// A time instance function block that represents a date and time value based on the Unix epoch (1st Jan 1970, 00:00:00.000).
// The block provides various methods and properties to interact with the time instance, including support for UTC and local time representations.
// It can be used for time calculations, comparisons, and conversions to different time formats (e.g., `DT`, `DATE`, `TOD`).
//
// [usage]
// The time instance can be set using various methods such as `FromDateTime` or `FromEpochMilliseconds`. 
// Use properties like `Year`, `Month`, `DayOfMonth`, `Hour`, and `Minute` to extract specific components of the date and time.
// Additionally, the `ToLocal` and `ToUTC` properties allow switching between different time modes.
// Use the `Kind` property to check the time mode.
{attribute 'enable_dynamic_creation'}
{attribute 'no_explicit_call' := 'calling this function block directly is not allowed'}
FUNCTION_BLOCK FINAL FB_TimeInstance 
IMPLEMENTS 
	I_TimeInstance, I_ComparableTimesInstance, I_EquatableTimesInstance, 
	I_TimeInstanceProperties, I_TimeInstanceArithmetics, I_TimeInstanceConversions
VAR
    _nEpochMilliseconds : ULINT; // The raw time instance value in milliseconds since 1st Jan 1970.
    _Date				: SysTimeRtc.SYSTIMEDATE; // Structured representation of the time instance (year, month, day, etc.).
    _eKind				: E_TimeInstanceKind; // Indicates whether the time instance is in UTC or Local time.
END_VAR

// The day of the month extracted from the time instance.
// [get] Returns the day component of the date, with a value ranging from 1 to 31.
PROPERTY DayOfMonth : T_DayOfMonth
GET
DayOfMonth := THIS^._Date.wDay;
END_GET
END_PROPERTY

// The day of the week extracted from the time instance.
// [get] Returns the day as an `E_DayOfWeek` enum or value ranging from 1 (Monday) to 7 (Sunday).
PROPERTY DayOfWeek : E_DayOfWeek
GET
DayOfWeek := THIS^._Date.wDayOfWeek;
END_GET
END_PROPERTY

// The day of the year extracted from the time instance.
// [get] Returns the day of the year, with a value ranging from 1 to 366.
PROPERTY DayOfYear : T_DayOfYear
GET
DayOfYear := THIS^._Date.wYday;
END_GET
END_PROPERTY

// The time instance value represented as the number of milliseconds since
// Thursday, 1.1.1970 00:00:00.000 (Unix epoch).
// [get] Returns the time instance value in milliseconds.
PROPERTY EpochMilliseconds : ULINT
GET
EpochMilliseconds := THIS^._nEpochMilliseconds;
END_GET
END_PROPERTY

// Sets the time instance based on a given `DATE` value as UTC.
METHOD FromDate : I_TimeInstance // A reference to the current instance.
VAR_INPUT
	// The input `DATE` value to convert to a time instance.
	dValue : DATE;
END_VAR
VAR_OUTPUT
	// Error code indicating the result of the operation.
	Error : FsError.T_Error;
END_VAR
FromDate := THIS^;

THIS^.FromEpochMilliseconds(TO_ULINT(dValue) * 1000, Error => Error);
END_METHOD

// Sets the time instance based on a given `DT` (Date and Time) value as UTC.
METHOD FromDateTime : I_TimeInstance // A reference to the current instance.
VAR_INPUT
	// The input `DT` value to convert to a time instance.
	dtValue : DT;
END_VAR
VAR_OUTPUT
	// Error code indicating the result of the operation.
	Error : FsError.T_Error;
END_VAR
FromDateTime := THIS^;

THIS^.FromEpochMilliseconds(TO_ULINT(dtValue) * 1000, Error => Error);
END_METHOD

// Sets the time instance based on a given number of milliseconds since the Unix epoch (1st Jan 1970, 00:00:00.000).
METHOD FromEpochMilliseconds : I_TimeInstance // A reference to the current instance.
VAR_INPUT
	// The input time instance value representing the number of milliseconds since 1st Jan 1970, 00:00:00.000.
	nValue : ULINT;
END_VAR
VAR_OUTPUT
	// Error code indicating the result of the operation.
	Error : FsError.T_Error;
END_VAR
VAR
	eResult : FsError.E_CodesysCmpError;
END_VAR
FromEpochMilliseconds := THIS^;

IF THIS^._nEpochMilliseconds = nValue THEN RETURN; END_IF

eResult := SysTimeRtc.SysTimeRtcConvertHighResToDate(nValue, THIS^._Date);
CASE eResult OF
	FsError.E_CodesysCmpError.ERR_OK:
		THIS^._eKind := E_TimeInstanceKind.UTC;
		THIS^._nEpochMilliseconds := nValue;
ELSE
	Error := 
		FsError.F_CreateErrorFromStartRange(
			FsError.GVL_ErrorDescriptors.fbGeneralErrorCodes,
			FsError.E_GeneralErrorCode.ERR_CODESYS_BEGIN,
			eResult);
	THIS^.FB_init(FALSE, FALSE);
	END_CASE
END_METHOD

// Sets the time instance using the specified `LTIME` value. 
// This method converts the input value to milliseconds since the Unix epoch (1st Jan 1970, 00:00:00.000). 
//
// [note] 
// The method only considers the time value down to the millisecond precision. 
// Any values smaller than 1ms (e.g., microseconds or nanoseconds) will be ignored.
METHOD FromTime : I_TimeInstance // A reference to the current instance.
VAR_INPUT
	// The time value to be set, provided as an LTIME datatype (milliseconds since the Unix epoch).
	tValue : LTIME;
END_VAR
VAR_OUTPUT
	// Error code indicating the result of the operation.
	Error : FsError.T_Error;
END_VAR
FromTime := THIS^;

THIS^.FromEpochMilliseconds(TO_ULINT(tValue) / TO_ULINT(LTIME#1MS), Error => Error);
END_METHOD

// Sets the time instance based on a given `TOD` (Time Of Day) value as UTC.
METHOD FromTimeOfDay : I_TimeInstance // A reference to the current instance.
VAR_INPUT
	// The input `TOD` value to convert to a time instance.
	tdValue : TOD;
END_VAR
VAR_OUTPUT
	// Error code indicating the result of the operation.
	Error : FsError.T_Error;
END_VAR
FromTimeOfDay := THIS^;

THIS^.FromEpochMilliseconds(TO_ULINT(tdValue), Error => Error);
END_METHOD

// The hour of the day extracted from the time instance.
// [get] Returns the hour component of the time, with a value ranging from 0 to 23.
PROPERTY Hour : T_Hour
GET
Hour := THIS^._Date.wHour;
END_GET
END_PROPERTY

// The reference to the current time instance.
// [get] Returns a reference to the current time instance implementing `I_TimeInstance`.
PROPERTY Instance : I_TimeInstance
GET
Instance := THIS^;
END_GET
END_PROPERTY

// Checks if the current time instance is after the specified time instance.
METHOD IsAfter : BOOL // TRUE if the current time instance is after the specified one, FALSE otherwise.
VAR_INPUT
	// The time instance to compare against.
	ipOther : I_TimeInstance;
END_VAR
IsAfter := 
	ipOther <> 0
	AND_THEN
	THIS^._nEpochMilliseconds > ipOther.EpochMilliseconds;
END_METHOD

// Checks if the current time instance is before the specified time instance.
METHOD IsBefore : BOOL // TRUE if the current time instance is before the specified one, FALSE otherwise.
VAR_INPUT
	// The time instance to compare against.
	ipOther : I_TimeInstance;
END_VAR
IsBefore := 
	ipOther <> 0
	AND_THEN
	THIS^._nEpochMilliseconds < ipOther.EpochMilliseconds;
END_METHOD

// Checks if the current time instance is equal to the specified time instance.
METHOD IsEqualTo : BOOL // TRUE if the current time instance is equal to the specified, FALSE otherwise.
VAR_INPUT
	// The time instance to compare against.
	ipOther : I_TimeInstance;
END_VAR
IsEqualTo := 
	ipOther <> 0
	AND_THEN
	THIS^._nEpochMilliseconds = ipOther.EpochMilliseconds;
END_METHOD

// Specifies whether the time instance is in UTC or local time format.
// [get] Returns the time instance type enum as a value.
PROPERTY Kind : E_TimeInstanceKind
GET
Kind := THIS^._eKind;
END_GET
END_PROPERTY

// The millisecond part of the second extracted from the time instance.
// [get] Returns the millisecond component, with a value ranging from 0 to 999.
PROPERTY Millisecond : T_Millisecond
GET
Millisecond := THIS^._Date.wMilliseconds;
END_GET
END_PROPERTY

// The minute of the hour extracted from the time instance.
// [get] Returns the minute component, with a value ranging from 0 to 59.
PROPERTY Minute : T_Minute
GET
Minute := THIS^._Date.wMinute;
END_GET
END_PROPERTY

// The month of the year extracted from the time instance.
// [get] Returns the month as an `E_Month` enum or a value ranging from 1 to 12 value.
PROPERTY Month : E_Month
GET
Month := THIS^._Date.wMonth;
END_GET
END_PROPERTY

// Updates the internal epoch milliseconds of the time instance to the current system time in UTC format.
METHOD Now : REFERENCE TO FB_TimeInstance // A reference to the current instance.
VAR_OUTPUT
	// Error code indicating the result of the operation.
	Error : FsError.T_Error;
END_VAR
VAR
	eResult : FsError.E_CodesysCmpError;
END_VAR
Now REF= THIS^;

// Get the current time instance as UTC.
eResult := SysTimeRtc.SysTimeRtcHighResGet(THIS^._nEpochMilliseconds);
CASE eResult OF
	FsError.E_CodesysCmpError.ERR_OK:
		SysTimeRtc.SysTimeRtcConvertHighResToDate(THIS^._nEpochMilliseconds, THIS^._Date);
ELSE // Reset the time instance class if there's an error.
	Error := 
		FsError.F_CreateErrorFromStartRange(
			FsError.GVL_ErrorDescriptors.fbGeneralErrorCodes,
			FsError.E_GeneralErrorCode.ERR_CODESYS_BEGIN,
			eResult);
	THIS^.FB_init(FALSE, FALSE);
	END_CASE
END_METHOD

// The second of the minute extracted from the time instance.
// [get] Returns the second component, with a value ranging from 0 to 59.
PROPERTY Second : T_Second
GET
Second := THIS^._Date.wSecond;
END_GET
END_PROPERTY

// Converts the time instance to a date value.
METHOD ToDate : DATE // The date part of the time instance.
VAR_OUTPUT
	// Error code indicating the result of the operation.
	Error : FsError.T_Error;
END_VAR
ToDate := TO_DATE(THIS^.ToDateTime(Error => Error));
END_METHOD

// Converts the time instance to a combined date and time value.
METHOD ToDateTime : DT // The combined date and time value as a DT (Date and Time).
VAR_OUTPUT
	// Error code indicating the result of the operation.
	Error : FsError.T_Error;
END_VAR
VAR
	nLocal : DWORD;
	eResult : FsError.E_CodesysCmpError;
END_VAR
CASE THIS^._eKind OF
	E_TimeInstanceKind.Local:
		eResult := SysTimeRtc.SysTimeRtcConvertUtcToLocal(
			TO_DWORD(THIS^._nEpochMilliseconds / 1000),
			nLocal);
	
		ToDateTime := TO_DT(nLocal);
		
		IF eResult <> FsError.E_CodesysCmpError.ERR_OK THEN 
			Error := 
				FsError.F_CreateErrorFromStartRange(
					FsError.GVL_ErrorDescriptors.fbGeneralErrorCodes,
					FsError.E_GeneralErrorCode.ERR_CODESYS_BEGIN,
					eResult);
			END_IF
		
ELSE 
	ToDateTime := TO_DT(THIS^._nEpochMilliseconds / 1000);
	END_CASE
END_METHOD

// Converts the time instance to local time representation.
METHOD ToLocal : I_TimeInstance // A reference to the current instance.
VAR_OUTPUT
	// Error code indicating the result of the operation.
	Error : FsError.T_Error;
END_VAR
VAR
	eResult : FsError.E_CodesysCmpError;
END_VAR
ToLocal := THIS^;

IF THIS^._eKind = E_TimeInstanceKind.Local THEN RETURN; END_IF;

eResult := SysTimeRtc.SysTimeRtcConvertHighResToLocal(THIS^._nEpochMilliseconds, THIS^._Date);
CASE eResult OF
	FsError.E_CodesysCmpError.ERR_OK:
		THIS^._eKind := E_TimeInstanceKind.Local;
ELSE
	Error := 
		FsError.F_CreateErrorFromStartRange(
			FsError.GVL_ErrorDescriptors.fbGeneralErrorCodes,
			FsError.E_GeneralErrorCode.ERR_CODESYS_BEGIN,
			eResult);
	END_CASE
END_METHOD

// Converts the time instance to a time of day  value.
METHOD ToTimeOfDay : TOD // The time of day part of the time instance.
VAR_INPUT
END_VAR
ToTimeOfDay := TO_TOD(
	(THIS^._Date.wHour * TO_DWORD(TOD#01:00:00.000))
	+
	(THIS^._Date.wMinute * TO_DWORD(TOD#00:01:00.000))
	+ 
	(THIS^._Date.wSecond * TO_DWORD(TOD#00:00:01.000))
	+ 
	THIS^._Date.wMilliseconds);
END_METHOD

// Converts the time instance to UTC time representation.
METHOD ToUTC : I_TimeInstance // A reference to the current instance.
VAR_OUTPUT
	// Error code indicating the result of the operation.
	Error : FsError.T_Error;
END_VAR
VAR
	eResult : FsError.E_CodesysCmpError;
END_VAR
ToUTC := THIS^;

IF THIS^._eKind = E_TimeInstanceKind.UTC THEN RETURN; END_IF;

eResult := SysTimeRtc.SysTimeRtcConvertHighResToDate(THIS^._nEpochMilliseconds, THIS^._Date);
CASE eResult OF
	FsError.E_CodesysCmpError.ERR_OK:
		THIS^._eKind := E_TimeInstanceKind.UTC;
ELSE
	Error := 
		FsError.F_CreateErrorFromStartRange(
			FsError.GVL_ErrorDescriptors.fbGeneralErrorCodes,
			FsError.E_GeneralErrorCode.ERR_CODESYS_BEGIN,
			eResult);
	END_CASE
END_METHOD

// The year extracted from the time instance.
// [get] Returns the year as a 4 digit value.
PROPERTY Year : T_Year
GET
Year := THIS^._Date.wYear;
END_GET
END_PROPERTY

END_FUNCTION_BLOCK

(* stored: Version 1.1.0.1
   POU FB_TimeInstance: Id {e6e6de43-7b7f-074b-1ca2-4b053bea74e2}, SpecialFunc None
   Property DayOfMonth: Id {60e816e1-4435-0612-1eae-4d7005c3d9fb}
   Get Get: Id {3907a527-b18e-0503-12be-c51e2dbc8e67}
   Property DayOfWeek: Id {59f79d25-beac-0bde-08ed-1040cb742c57}
   Get Get: Id {8d78e11e-55dc-0c40-3dde-ce876e3fb30b}
   Property DayOfYear: Id {362b65ee-c21c-0c53-03d9-e3bf2606a66b}
   Get Get: Id {e762102a-48dc-019e-127f-fd4d88b185cc}
   Property EpochMilliseconds: Id {20301beb-082b-097b-1c4e-628b84fa049a}
   Get Get: Id {7077aa0d-dfac-05c6-3c0e-51fb09ce5e0b}
   Method FromDate: Id {42e1dd4b-64bc-0652-35b6-11c170ba588f}
   Method FromDateTime: Id {ccb59f48-60a9-0163-3fe2-e66c66b0578d}
   Method FromEpochMilliseconds: Id {981d420c-033f-01b4-325c-9d1f4c94167f}
   Method FromTime: Id {fe00b6a2-8466-0e34-2dac-d4faeee2cf7f}
   Method FromTimeOfDay: Id {cc6108ea-0cc3-0982-0207-ff06faa4e04b}
   Property Hour: Id {90138cb2-1221-0609-030d-4f9ef31dc45c}
   Get Get: Id {37588880-29d2-0e46-311f-356406dc721c}
   Property Instance: Id {69ebd0df-325d-02f3-13a8-a8969e45adc2}
   Get Get: Id {b6878157-2ede-0255-25ee-95c0daf56b49}
   Method IsAfter: Id {2cae66b8-d1e7-0d00-329c-004410e04b9c}
   Method IsBefore: Id {7bdfa8a4-9e8c-08f7-2a9e-dd667eefde6f}
   Method IsEqualTo: Id {dba8a7a0-0fb8-0377-3898-12345927eed2}
   Property Kind: Id {658eca20-c9a9-0a35-0410-abd3c3bb0096}
   Get Get: Id {c8271b94-a3ea-0898-3d8d-3bce821625da}
   Property Millisecond: Id {08face5a-d595-0366-1b6e-3949928e1e48}
   Get Get: Id {a2f4f72b-afe3-069a-099b-63ebd77733e5}
   Property Minute: Id {15bbdfde-68d3-0477-1d1a-e9c08dbf3a01}
   Get Get: Id {2f040977-7fbf-0347-26fe-85d0654f570f}
   Property Month: Id {62c0f3ed-8996-053c-1c72-3a5c119d406a}
   Get Get: Id {7d094cda-b6c5-0b42-1c78-04bd7a82240a}
   Method Now: Id {b1bf1f77-5c7b-0d28-1300-c411e2b5f387}
   Property Second: Id {59b40d1c-5d89-06ad-2653-2b8aac68b854}
   Get Get: Id {25a59e15-b6b3-0bc0-1fe3-38390475049f}
   Method ToDate: Id {d572272b-a7aa-08b5-0c53-7ec2690a611f}
   Method ToDateTime: Id {4f912b94-33c5-05cd-0495-31634f7ea87d}
   Method ToLocal: Id {fc041b72-7528-0bf2-2775-d53fe075b280}
   Method ToTimeOfDay: Id {b154d6aa-ef4e-0f4d-2d55-601e4067cc63}
   Method ToUTC: Id {284b9878-067f-0ffc-19c1-27df0a954c5d}
   Property Year: Id {90baf8ce-ec87-0268-21c2-f6aa6f365dda}
   Get Get: Id {c459bc70-ad56-0fea-34d6-c0f0cb921b1f} *)
